(* IEC 61131-3 sources: POMIRTS_lab3/AS/Library_2/AsNxCoS, 3 files *)

(* ---- AsNxCoS.typ ---- *)
TYPE

END_TYPE

(* ---- AsNxCoS.fun ---- *)
{REDUND_CONTEXT} {REDUND_UNREPLICABLE} FUNCTION_BLOCK nxcosNmt					(*send NMT command*)
	VAR_INPUT
		enable			: BOOL;			(*enables execution*)
		pDevice			: UDINT;		(*interface name given as a pointer, e.g., "SL<x>.SS<y>.IF<z>"*)
		command			: UDINT;		(*NMT command*)
	END_VAR
	VAR
        _state			: UINT;			(*internal variable*)
		_result			: UINT;			(*internal variable*)
        _srcId			: UDINT;		(*internal variable*)
	END_VAR
	VAR_OUTPUT
		status			: UINT;			(*execution status: ERR_OK, ERR_FUB_ENABLE_FALSE, ERR_FUB_BUSY, 0xXXXX = see help*)
		coStatus		: UDINT;		(*CANopen stack status*)
	END_VAR
END_FUNCTION_BLOCK

{REDUND_CONTEXT} {REDUND_UNREPLICABLE} FUNCTION_BLOCK nxcosStartStop			(*start/stop CANopen bus slave*)
	VAR_INPUT
		enable			: BOOL;			(*enables execution*)
		pDevice			: UDINT;		(*interface name given as a pointer, e.g., "SL<x>.SS<y>.IF<z>"*)
		mode			: UDINT;		(*mode 0 = stop/ 1 = start*)
	END_VAR
	VAR
        _state			: UINT;			(*internal variable*)
		_result			: UINT;			(*internal variable*)
        _srcId			: UDINT;		(*internal variable*)
	END_VAR
	VAR_OUTPUT
		status			: UINT;			(*execution status: ERR_OK, ERR_FUB_ENABLE_FALSE, ERR_FUB_BUSY, 0xXXXX = see help*)
		coStatus		: UDINT;		(*CANopen stack status*)
	END_VAR
END_FUNCTION_BLOCK

{REDUND_CONTEXT} {REDUND_UNREPLICABLE} FUNCTION_BLOCK nxcosWriteEmcy			(*write emergency telegrams*)
	VAR_INPUT
		enable			: BOOL;			(*enables execution*)
		pDevice			: UDINT;		(*interface name given as a pointer, e.g., "SL<x>.SS<y>.IF<z>"*)
		errorCode		: UINT;			(*error code*)
		errorRegister	: USINT;		(*error register*)
		pManErrorCode	: UDINT;		(*man error code given as pointer*)
	END_VAR
	VAR
        _state			: UINT;			(*internal variable*)
		_result			: UINT;			(*internal variable*)
        _srcId			: UDINT;		(*internal variable*)
	END_VAR
	VAR_OUTPUT
		status			: UINT;			(*execution status: ERR_OK, ERR_FUB_ENABLE_FALSE, ERR_FUB_BUSY, 0xXXXX = see help*)
		coStatus		: UDINT;		(*CANopen stack status*)
	END_VAR
END_FUNCTION_BLOCK

{REDUND_CONTEXT} {REDUND_UNREPLICABLE} FUNCTION_BLOCK nxcosSetAdr				(*set address*)
	VAR_INPUT
		enable			: BOOL;			(*enables execution*)
		pDevice			: UDINT;		(*interface name given as a pointer, e.g., "SL<x>.SS<y>.IF<z>"*)
		address			: UDINT;		(*new slave address*)
	END_VAR
	VAR
        _state			: UINT;			(*internal variable*)
		_result			: UINT;			(*internal variable*)
        _srcId			: UDINT;		(*internal variable*)
	END_VAR
	VAR_OUTPUT
		status			: UINT;			(*execution status: ERR_OK, ERR_FUB_ENABLE_FALSE, ERR_FUB_BUSY, 0xXXXX = see help*)
		coStatus		: UDINT;		(*CANopen stack status*)
	END_VAR
END_FUNCTION_BLOCK

{REDUND_CONTEXT} {REDUND_UNREPLICABLE} FUNCTION_BLOCK nxcosStartBusComm		(*start bus communication*)
	VAR_INPUT
		enable			: BOOL;			(*enables execution*)
		pDevice			: UDINT;		(*interface name given as a pointer, e.g., "SL<x>.SS<y>.IF<z>"*)
	END_VAR
	VAR
        _state			: UINT;			(*internal variable*)
		_result			: UINT;			(*internal variable*)
        _srcId			: UDINT;		(*internal variable*)
	END_VAR
	VAR_OUTPUT
		status			: UINT;			(*execution status: ERR_OK, ERR_FUB_ENABLE_FALSE, ERR_FUB_BUSY, 0xXXXX = see help*)
		coStatus		: UDINT;		(*CANopen stack status*)
	END_VAR
END_FUNCTION_BLOCK

(* ---- AsNxCoS.var ---- *)
VAR CONSTANT
	nxcosERR_INVALID_DEVICE					: UINT	:= 34600;	(*error invalid device*)
	nxcosERR_SEND_MESSAGE					: UINT	:= 34601;	(*error send message*)
	nxcosERR_TIMEOUT						: UINT	:= 34602;	(*error timeout*)
	nxcosERR_CANOPEN_STACK					: UINT	:= 34603;	(*error receive message*)
	nxcosERR_PARAMETER						: UINT	:= 34604;	(*error invalid parameter*)

	nxcosNMT_CMD_START						: UDINT	:= 1;		(*start the node*)
	nxcosNMT_CMD_STOP						: UDINT	:= 2;		(*stop the node*)
	nxcosNMT_CMD_ENTER_PREOP				: UDINT	:= 128;		(*set the node into the pre-operational mode*)
	nxcosNMT_CMD_RESET_NODE					: UDINT	:= 129;		(*reset the node*)
	nxcosNMT_CMD_RESET_COMM					: UDINT	:= 130;		(*reset the communication to the node*)

	nxcosMODE_STOP							: UDINT := 0;		(*mode stop*)
	nxcosMODE_START							: UDINT := 1;		(*mode start*)

	nxcosEREG_ERROR_RESET					: USINT := 16#00;
	nxcosEREG_GENERIC_BIT					: USINT := 16#01;
	nxcosEREG_CURRENT_BIT					: USINT := 16#02;
	nxcosEREG_VOLTAGE_BIT					: USINT := 16#04;
	nxcosEREG_TEMPERATURE_BIT				: USINT := 16#08;
	nxcosEREG_COMM_ERROR_BIT				: USINT := 16#10;
	nxcosEREG_DEV_PROFILE_BIT				: USINT := 16#20;
	nxcosEREG_MANU_SPEC_BIT					: USINT := 16#80;
END_VAR
